// TwinCAT 3 PLC project PLC
// Title: TcControls
// Company: inspire AG
// Author: Roald Ruiter
// ProjectVersion: 0.1.0
// Description: PID control function blocks
// ProgramVersion: 3.1.4023.0
// libraries:
//   Tc3_Module, * (Beckhoff Automation GmbH)
//   TcUnit, * (www.tcunit.org)
// project tree:
//   / Pid.TcPOU, IPid.TcIO, PidParameters.TcDUT (not stored), PlcTask.TcTTO (not stored)
//   Tests/ Pid_Tests.TcPOU, UnitTests.TcPOU
// real-time tasks:
//   TASK PlcTask: cycle T#10ms, priority 21, ADS port 351

// ---- IPid.TcIO
INTERFACE IPid

PROPERTY Out : LREAL
GET
END_GET
END_PROPERTY

PROPERTY PreviousIntegralPart : LREAL
SET
END_SET
END_PROPERTY

END_INTERFACE

// ---- Pid.TcPOU
FUNCTION_BLOCK Pid IMPLEMENTS IPid
VAR_INPUT
    setpoint : LREAL;
    actual : LREAL;
    parameters : PidParameters;
END_VAR
VAR
    _error : LREAL;
    _previousError : LREAL;
    _deltaError : LREAL;
    _proportionalPart : LREAL;
    _integralPart : LREAL;
    _previousIntegralPart : LREAL;
    _differentialPart : LREAL;
    _differentialPartLimit : LREAL;
    _out : LREAL;
END_VAR

_error := setpoint - actual;

_proportionalPart := parameters.Kp * _error;

_integralPart := _previousIntegralPart + parameters.Ki * _error;
_previousIntegralPart := _integralPart;

_deltaError := _error - _previousError;
IF _differentialPartLimit = 0 OR _deltaError <= _differentialPartLimit THEN
    _differentialPart := _deltaError * parameters.Kd;
END_IF
_previousError := _error;

_out := _proportionalPart + _integralPart + _differentialPart;

PROPERTY DifferentialPartLimit : LREAL
SET
_differentialPartLimit := DifferentialPartLimit;
END_SET
END_PROPERTY

PROPERTY Out : LREAL
GET
Out := _out;
END_GET
END_PROPERTY

PROPERTY PreviousIntegralPart : LREAL
SET
_previousIntegralPart := PreviousIntegralPart;
END_SET
END_PROPERTY

END_FUNCTION_BLOCK

// ---- Tests/Pid_Tests.TcPOU
FUNCTION_BLOCK Pid_Tests EXTENDS FB_TestSuite
VAR
    delta : LREAL := 1E-5;
END_VAR

OnlyProportionalPart();
OnlyPropotionalPartRunTwiceWithDifferentInputs();
OnlyIntegralPart();
OnlyIntegralPartSetPreviousIntegralPartBefore();
OnlyDifferentialPart();
OnlyDifferentialPartWithDiffLimit();

METHOD OnlyDifferentialPart
VAR_INST
    P : Pid;
    parameters : PidParameters := (Kd:=0.01);
END_VAR
TcUnit.TEST('OnlyDifferentialPart');

P(setpoint:=10, actual:=6, parameters:=parameters);
AssertEquals_LREAL(
    Expected:=0.04,
    Actual:=P.Out,
    Delta:=delta,
    Message:='Pid output run 1 not correct'
);

P(setpoint:=10, actual:=8, parameters:=parameters);
AssertEquals_LREAL(
    Expected:=-0.02,
    Actual:=P.Out,
    Delta:=delta,
    Message:='Pid output run 2 not correct'
);

TcUnit.TEST_FINISHED();
END_METHOD

METHOD OnlyDifferentialPartWithDiffLimit
VAR_INST
    P : Pid;
    parameters : PidParameters := (Kd:=0.01);
END_VAR
TcUnit.TEST('OnlyDifferentialPartWithDiffLimit');

P.DifferentialPartLimit := 3;
P(setpoint:=10, actual:=6, parameters:=parameters);
AssertEquals_LREAL(
    Expected:=0,
    Actual:=P.Out,
    Delta:=delta,
    Message:='Pid output run 1 not correct'
);

P(setpoint:=10, actual:=8, parameters:=parameters);
AssertEquals_LREAL(
    Expected:=-0.02,
    Actual:=P.Out,
    Delta:=delta,
    Message:='Pid output run 2 not correct'
);

TcUnit.TEST_FINISHED();
END_METHOD

METHOD OnlyIntegralPart
VAR_INST
    P : Pid;
    parameters : PidParameters := (Ki:=0.25);
END_VAR
TcUnit.TEST('OnlyIntegralPart');

P(setpoint:=10, actual:=6, parameters:=parameters);
AssertEquals_LREAL(
    Expected:=1,
    Actual:=P.Out,
    Delta:=delta,
    Message:='Pid output run 1 not correct'
);

P(setpoint:=10, actual:=8, parameters:=parameters);
AssertEquals_LREAL(
    Expected:=1.5,
    Actual:=P.Out,
    Delta:=delta,
    Message:='Pid output run 2 not correct'
);

TcUnit.TEST_FINISHED();
END_METHOD

METHOD OnlyIntegralPartSetPreviousIntegralPartBefore
VAR_INST
    P : Pid;
    parameters : PidParameters := (Ki:=0.25);
END_VAR
TcUnit.TEST('OnlyIntegralPartSetPreviousIntegralPartBefore');

P.PreviousIntegralPart := 3;

P(setpoint:=10, actual:=6, parameters:=parameters);
AssertEquals_LREAL(
    Expected:=4,
    Actual:=P.Out,
    Delta:=delta,
    Message:='Pid output run 1 not correct'
);

P(setpoint:=10, actual:=8, parameters:=parameters);
AssertEquals_LREAL(
    Expected:=4.5,
    Actual:=P.Out,
    Delta:=delta,
    Message:='Pid output run 2 not correct'
);

TcUnit.TEST_FINISHED();
END_METHOD

METHOD OnlyProportionalPart
VAR_INST
    P : Pid;
    parameters : PidParameters := (Kp:=5);
END_VAR
TcUnit.TEST('OnlyProportionalPart');

P(setpoint:=10, actual:=5, parameters:=parameters);

AssertEquals_LREAL(Expected:=25, Actual:=P.Out, Delta:=delta, Message:='Pid output not correct');

TcUnit.TEST_FINISHED();
END_METHOD

METHOD OnlyPropotionalPartRunTwiceWithDifferentInputs
VAR_INST
    P : Pid;
    parameters : PidParameters := (Kp:=2);
END_VAR
TcUnit.TEST('OnlyPropotionalPartRunTwiceWithDifferentInputs');

P(setpoint:=3, actual:=4.5, parameters:=parameters);

AssertEquals_LREAL(
    Expected:=-3,
    Actual:=P.Out,
    Delta:=delta,
    Message:='Pid output after run 1 not correct'
);

P(setpoint:=-8, actual:=-6, parameters:=parameters);

AssertEquals_LREAL(
    Expected:=-4,
    Actual:=P.Out,
    Delta:=delta,
    Message:='Pid output after run 2 not correct'
);

TcUnit.TEST_FINISHED();
END_METHOD

END_FUNCTION_BLOCK

// ---- Tests/UnitTests.TcPOU
PROGRAM UnitTests
VAR
    pidTests : Pid_Tests;
END_VAR

TcUnit.RUN();

END_PROGRAM
